(* IEC 61131-3 sources: stverif/testfiles/Blackbox/src, 2 files *)

(* ---- function.fun ---- *)
FUNCTION Func : INT
    VAR_INPUT
        varx : INT;
    END_VAR
END_FUNCTION

(* ---- variables.var ---- *)
VAR
	a : INT;
	b : INT;
	c : REAL;
	d : INT;
	x : INT;
	y : REAL;
END_VAR
